FUNCTION_BLOCK StateCheck_View
  (* Version 0.1, 2005-12-14, Oscar Ljungkrantz, Chalmers *)
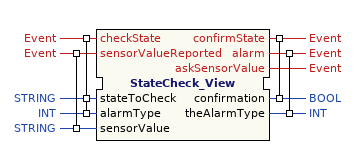
  EVENT_INPUT
    checkState WITH stateToCheck, alarmType;
    sensorValueReported WITH sensorValue;
  END_EVENT
  EVENT_OUTPUT
    confirmState WITH confirmation;
    alarm WITH theAlarmType;
    askSensorValue;
  END_EVENT
  VAR_INPUT
    stateToCheck : STRING;
    alarmType : INT;
    sensorValue : STRING;
  END_VAR
  VAR_OUTPUT
    confirmation : BOOL;
    theAlarmType : INT;
  END_VAR
  VAR
    currentStateToCheck : STRING;
    setAlarm : BOOL := FALSE;
    currentAlarmType : INT := 1;
  END_VAR
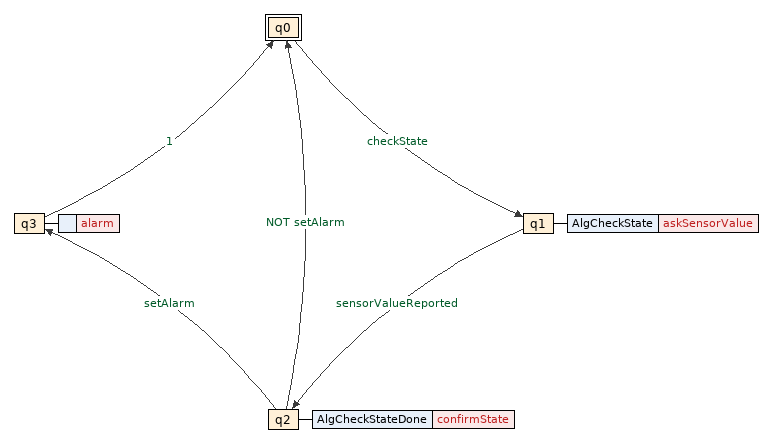
  EC_STATES
    q0;
    q1 : AlgCheckState -> askSensorValue;
    q2 : AlgCheckStateDone -> confirmState;
    q3 : -> alarm;
  END_STATES
  EC_TRANSITIONS
    q0 TO q1 := checkState;
    q1 TO q2 := sensorValueReported;
    q2 TO q3 := setAlarm;
    q2 TO q0 := NOT setAlarm;
    q3 TO q0 := 1;
  END_TRANSITIONS
  ALGORITHM AlgCheckState IN Java:
		currentStateToCheck = stateToCheck;
		currentAlarmType = alarmType;
  END_ALGORITHM
  ALGORITHM AlgCheckStateDone IN Java:
		if (sensorValue == currentStateToCheck)
		{
			confirmation = TRUE;
			setAlarm = FALSE;
		}
		else
		{
			confirmation = FALSE;
			setAlarm = TRUE;
			theAlarmType = currentAlarmType;
		}
  END_ALGORITHM
END_FUNCTION_BLOCK
